Staubli VAL3: getSize.pgx

public program getSize(num& x_nSize[], num x_nType)
begin
  // get the size of the Start list
  switch x_nType
    case 0
      // get the size of the Start list
      if saveCycle:sLoadStart!=""
        x_nSize=size(saveCycle:sLoadStart)
      else
        x_nSize=0
      endIf
    break
    case 1
      if saveCycle:sLoadProg!=""
        // get the size of the process list
        x_nSize=size(saveCycle:sLoadProg)
      else
        x_nSize=0
      endIf
    break
    case 2
      if saveCycle:sLoadEnd!=""
        // get the size of the End list
        x_nSize=size(saveCycle:sLoadEnd)
      else
        x_nSize=0
      endIf
    break
  endSwitch
end
